{attribute 'qualified_only'}
VAR_GLOBAL
	sPistonEndStopMessage : STRING;
	fCylinderPositonReference : LREAL := 0.0;
	fCylinderVelocityReference : LREAL := 0.0;
	eCraneStatus : E_CraneStatus;
	eCraneMode : E_CraneMode;
	
	fBoomAngle : LREAL;
	stAngleRelativeMovement : ST_RelativeMovement;
	
	bPower : BOOL;
	bStart : BOOL;
	bStop : BOOL;
	bRunning : BOOL := FALSE;
	bError : BOOL;
	bMode : BOOL;
END_VAR

(* stored: Version 1.1.0.1, ProductVersion 3.1.4024.10
   GVL HMI: Id {631d78cb-73d2-40fd-ac8b-c4cc47a6d8ff} *)
